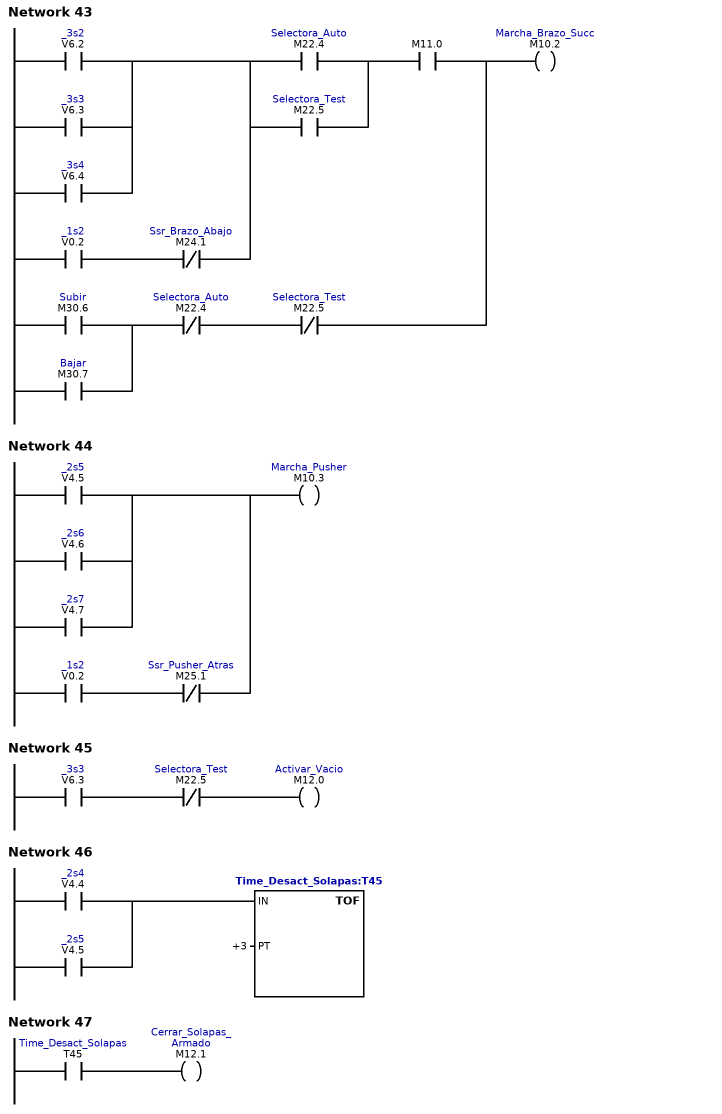
[picture p24: SBR6 networks 43-47]
Network 43
LD     _3s2:V6.2
O      _3s3:V6.3
O      _3s4:V6.4
LD     _1s2:V0.2
AN     Ssr_Brazo_Abajo:M24.1
OLD
LD     Selectora_Auto:M22.4
O      Selectora_Test:M22.5
ALD
A      M11.0
LD     Subir:M30.6
O      Bajar:M30.7
AN     Selectora_Auto:M22.4
AN     Selectora_Test:M22.5
OLD
=      Marcha_Brazo_Succ:M10.2
Network 44
LD     _2s5:V4.5
O      _2s6:V4.6
O      _2s7:V4.7
LD     _1s2:V0.2
AN     Ssr_Pusher_Atras:M25.1
OLD
=      Marcha_Pusher:M10.3
Network 45
LD     _3s3:V6.3
AN     Selectora_Test:M22.5
=      Activar_Vacio:M12.0
Network 46
LD     _2s4:V4.4
O      _2s5:V4.5
TOF    Time_Desact_Solapas:T45, +3
Network 47
LD     Time_Desact_Solapas:T45
=      Cerrar_Solapas_Armado:M12.1
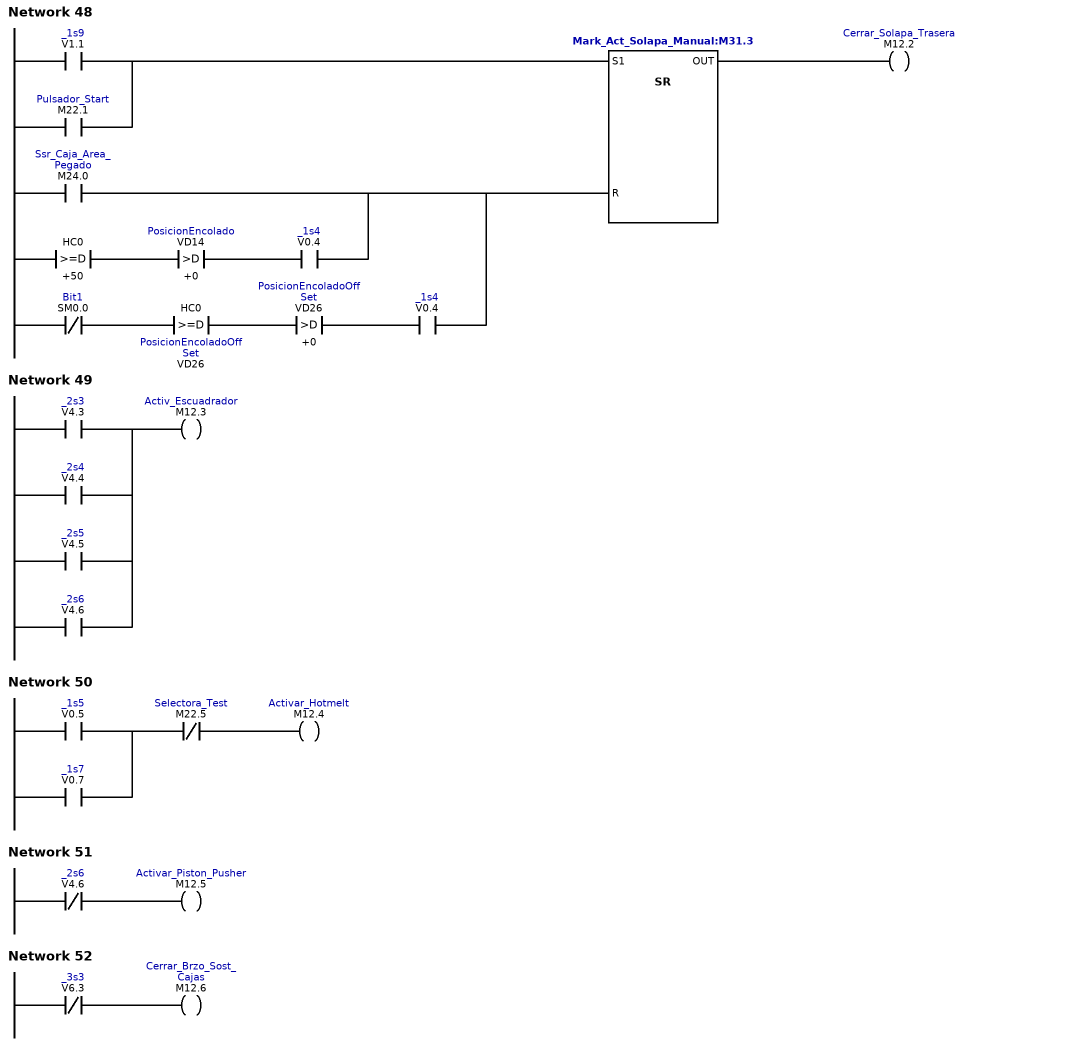
Network 48
LD     _1s9:V1.1
O      Pulsador_Start:M22.1
LD     Ssr_Caja_Area_Pegado:M24.0
LDD>=  HC0, +50
AD>    PosicionEncolado:VD14, +0
A      _1s4:V0.4
OLD
LDN    Bit1:SM0.0
AD>=   HC0, PosicionEncoladoOffSet:VD26
AD>    PosicionEncoladoOffSet:VD26, +0
A      _1s4:V0.4
OLD
NOT
A      Mark_Act_Solapa_Manual:M31.3
OLD
=      Mark_Act_Solapa_Manual:M31.3
=      Cerrar_Solapa_Trasera:M12.2
Network 49
LD     _2s3:V4.3
O      _2s4:V4.4
O      _2s5:V4.5
O      _2s6:V4.6
=      Activ_Escuadrador:M12.3
Network 50
LD     _1s5:V0.5
O      _1s7:V0.7
AN     Selectora_Test:M22.5
=      Activar_Hotmelt:M12.4
Network 51
LDN    _2s6:V4.6
=      Activar_Piston_Pusher:M12.5
Network 52
LDN    _3s3:V6.3
=      Cerrar_Brzo_Sost_Cajas:M12.6
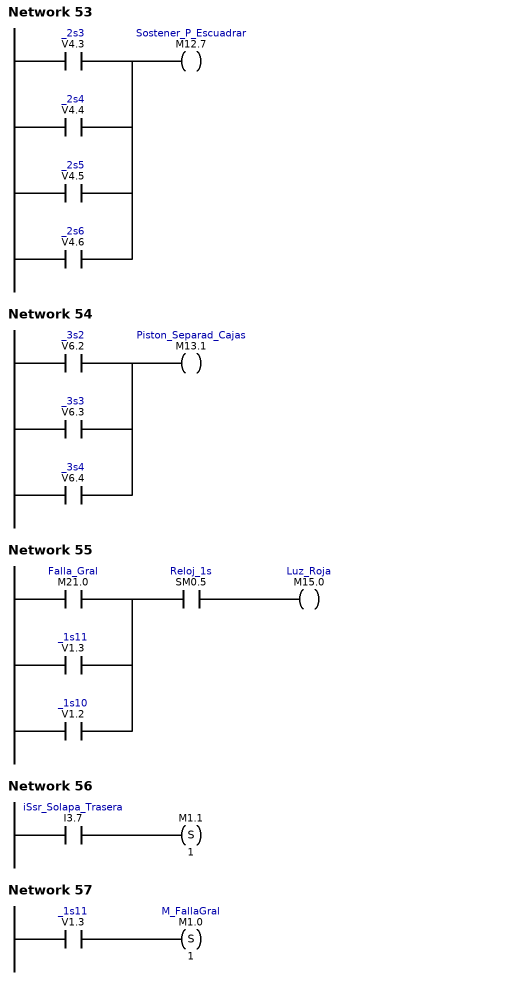
Network 53
LD     _2s3:V4.3
O      _2s4:V4.4
O      _2s5:V4.5
O      _2s6:V4.6
=      Sostener_P_Escuadrar:M12.7
Network 54
LD     _3s2:V6.2
O      _3s3:V6.3
O      _3s4:V6.4
=      Piston_Separad_Cajas:M13.1
Network 55
LD     Falla_Gral:M21.0
O      _1s11:V1.3
O      _1s10:V1.2
A      Reloj_1s:SM0.5
=      Luz_Roja:M15.0
Network 56
LD     iSsr_Solapa_Trasera:I3.7
S      M1.1, 1
Network 57
LD     _1s11:V1.3
S      M_FallaGral:M1.0, 1
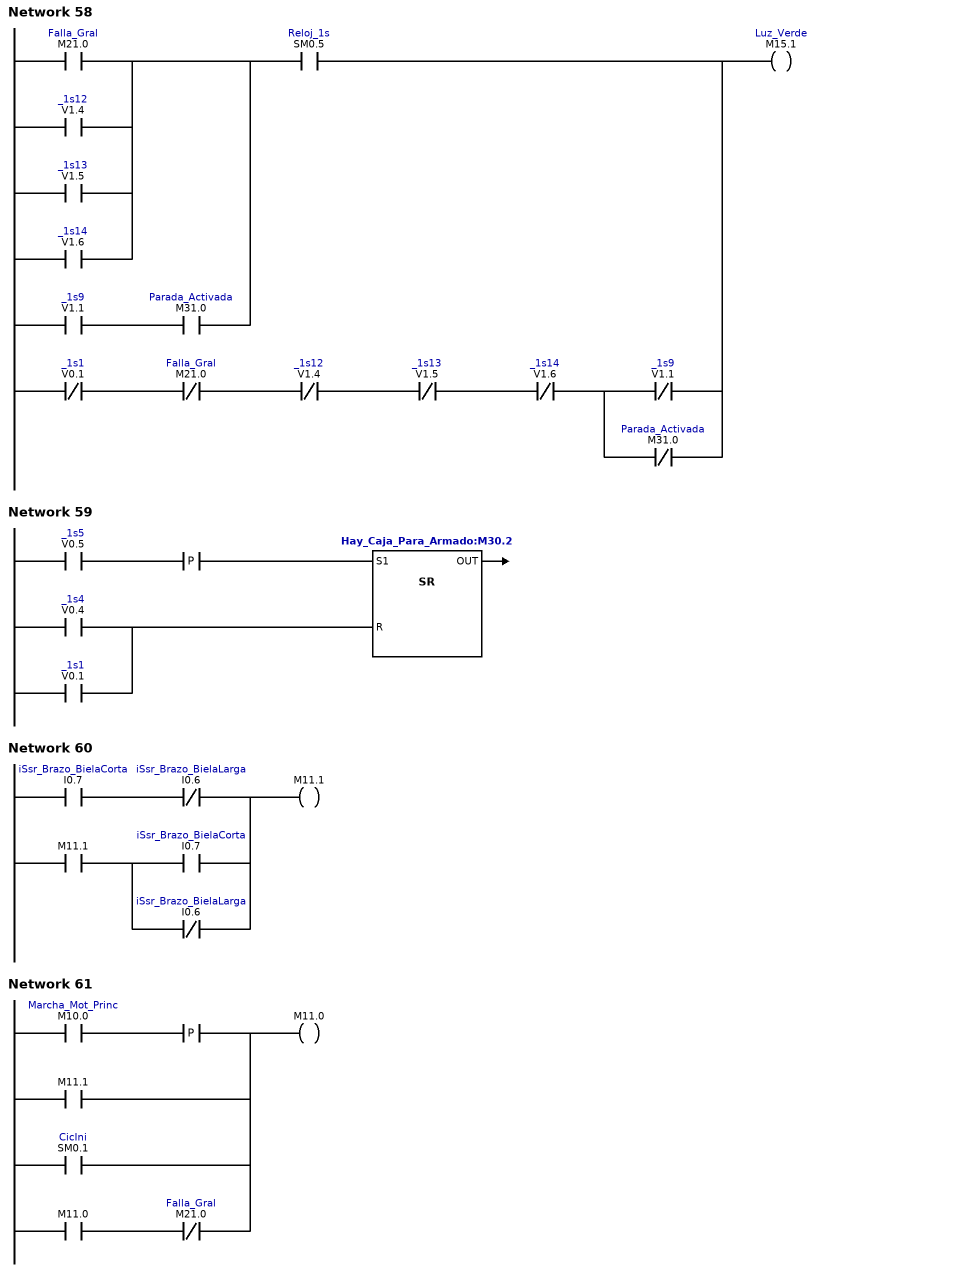
Network 58
LD     Falla_Gral:M21.0
O      _1s12:V1.4
O      _1s13:V1.5
O      _1s14:V1.6
LD     _1s9:V1.1
A      Parada_Activada:M31.0
OLD
A      Reloj_1s:SM0.5
LDN    _1s1:V0.1
AN     Falla_Gral:M21.0
AN     _1s12:V1.4
AN     _1s13:V1.5
AN     _1s14:V1.6
LDN    _1s9:V1.1
ON     Parada_Activada:M31.0
ALD
OLD
=      Luz_Verde:M15.1
Network 59
LD     _1s5:V0.5
EU
LD     _1s4:V0.4
O      _1s1:V0.1
NOT
A      Hay_Caja_Para_Armado:M30.2
OLD
=      Hay_Caja_Para_Armado:M30.2
Network 60
LD     iSsr_Brazo_BielaCorta:I0.7
AN     iSsr_Brazo_BielaLarga:I0.6
LD     M11.1
LD     iSsr_Brazo_BielaCorta:I0.7
ON     iSsr_Brazo_BielaLarga:I0.6
ALD
OLD
=      M11.1
Network 61
LD     Marcha_Mot_Princ:M10.0
EU
O      M11.1
O      CicIni:SM0.1
LD     M11.0
AN     Falla_Gral:M21.0
OLD
=      M11.0
END_SUBROUTINE_BLOCK

SUBROUTINE_BLOCK Secuencial_2:SBR7
TITLE=
BEGIN
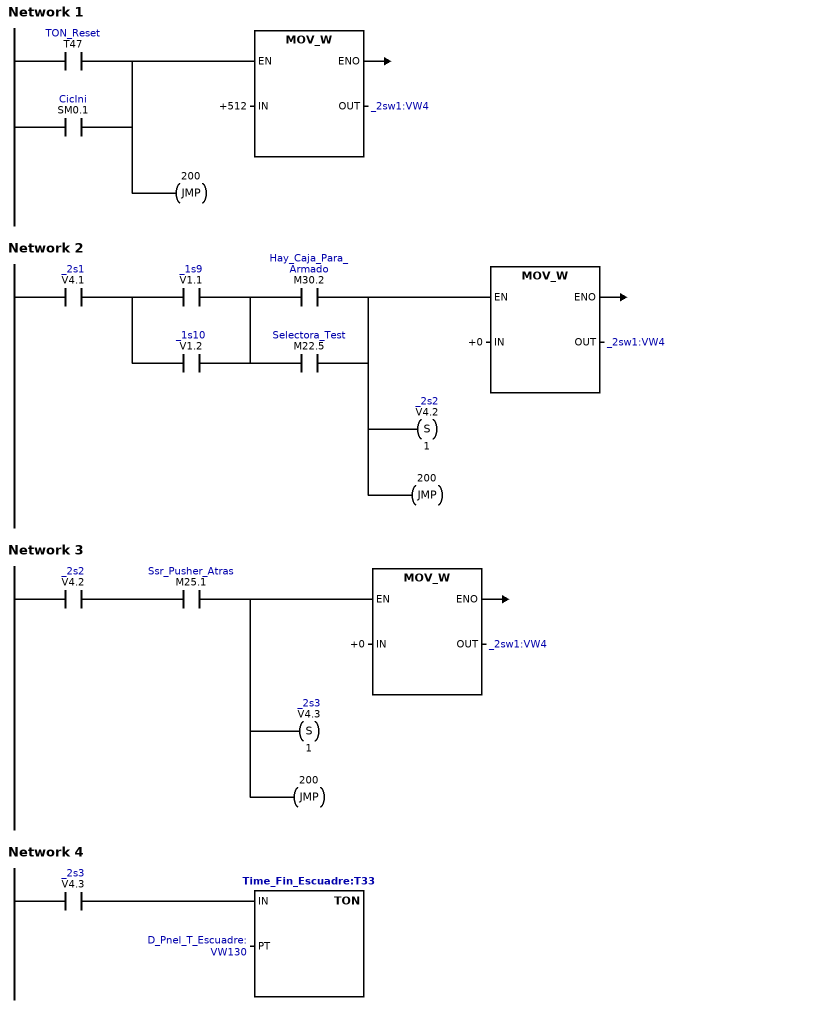
Network 1
LD     TON_Reset:T47
O      CicIni:SM0.1
MOVW   +512, _2sw1:VW4
JMP    200
Network 2
LD     _2s1:V4.1
LD     _1s9:V1.1
O      _1s10:V1.2
ALD
LD     Hay_Caja_Para_Armado:M30.2
O      Selectora_Test:M22.5
ALD
MOVW   +0, _2sw1:VW4
S      _2s2:V4.2, 1
JMP    200
Network 3
LD     _2s2:V4.2
A      Ssr_Pusher_Atras:M25.1
MOVW   +0, _2sw1:VW4
S      _2s3:V4.3, 1
JMP    200
Network 4
LD     _2s3:V4.3
TON    Time_Fin_Escuadre:T33, D_Pnel_T_Escuadre:VW130
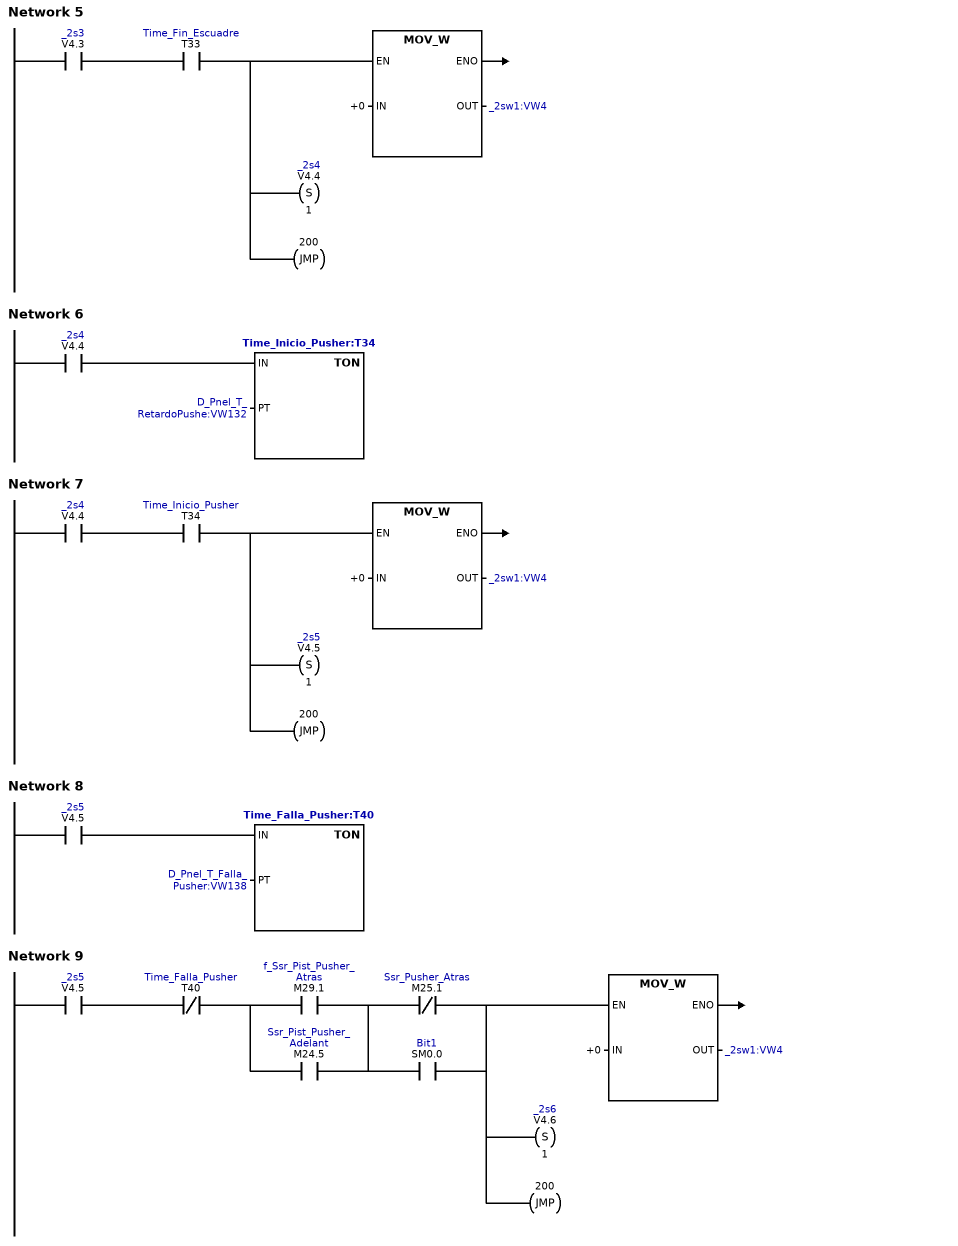
Network 5
LD     _2s3:V4.3
A      Time_Fin_Escuadre:T33
MOVW   +0, _2sw1:VW4
S      _2s4:V4.4, 1
JMP    200
Network 6
LD     _2s4:V4.4
TON    Time_Inicio_Pusher:T34, D_Pnel_T_RetardoPushe:VW132
Network 7
LD     _2s4:V4.4
A      Time_Inicio_Pusher:T34
MOVW   +0, _2sw1:VW4
S      _2s5:V4.5, 1
JMP    200
Network 8
LD     _2s5:V4.5
TON    Time_Falla_Pusher:T40, D_Pnel_T_Falla_Pusher:VW138
Network 9
LD     _2s5:V4.5
AN     Time_Falla_Pusher:T40
LD     f_Ssr_Pist_Pusher_Atras:M29.1
O      Ssr_Pist_Pusher_Adelant:M24.5
ALD
LDN    Ssr_Pusher_Atras:M25.1
O      Bit1:SM0.0
ALD
MOVW   +0, _2sw1:VW4
S      _2s6:V4.6, 1
JMP    200
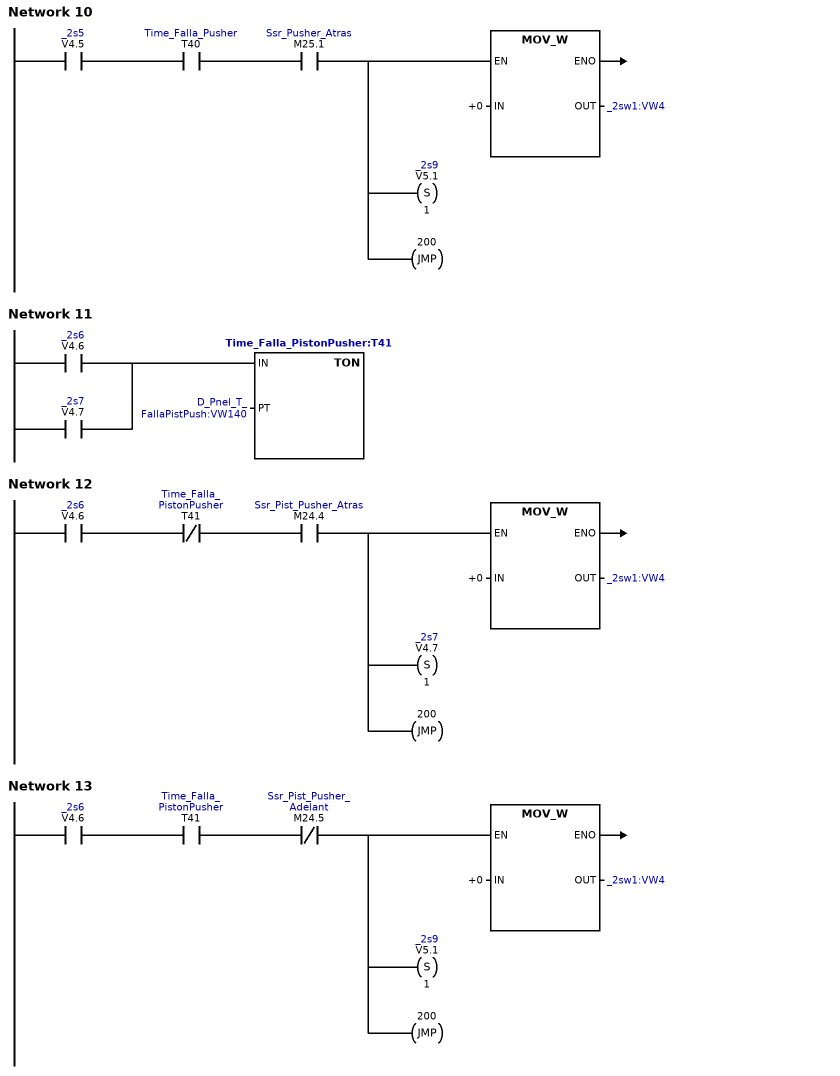
Network 10
LD     _2s5:V4.5
A      Time_Falla_Pusher:T40
A      Ssr_Pusher_Atras:M25.1
MOVW   +0, _2sw1:VW4
S      _2s9:V5.1, 1
JMP    200
Network 11
LD     _2s6:V4.6
O      _2s7:V4.7
TON    Time_Falla_PistonPusher:T41, D_Pnel_T_FallaPistPush:VW140
Network 12
LD     _2s6:V4.6
AN     Time_Falla_PistonPusher:T41
A      Ssr_Pist_Pusher_Atras:M24.4
MOVW   +0, _2sw1:VW4
S      _2s7:V4.7, 1
JMP    200
Network 13
LD     _2s6:V4.6
A      Time_Falla_PistonPusher:T41
AN     Ssr_Pist_Pusher_Adelant:M24.5
MOVW   +0, _2sw1:VW4
S      _2s9:V5.1, 1
JMP    200
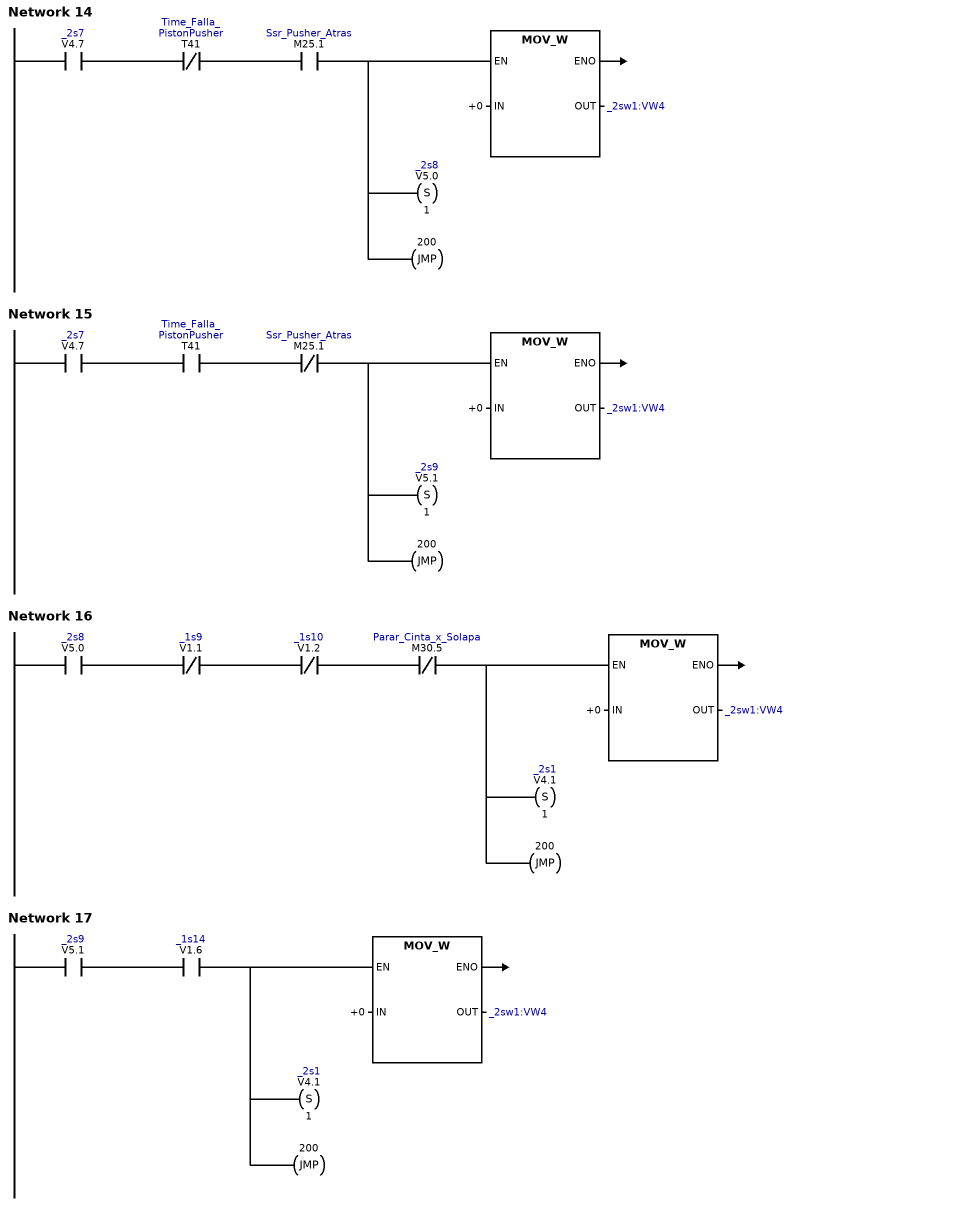
Network 14
LD     _2s7:V4.7
AN     Time_Falla_PistonPusher:T41
A      Ssr_Pusher_Atras:M25.1
MOVW   +0, _2sw1:VW4
S      _2s8:V5.0, 1
JMP    200
Network 15
LD     _2s7:V4.7
A      Time_Falla_PistonPusher:T41
AN     Ssr_Pusher_Atras:M25.1
MOVW   +0, _2sw1:VW4
S      _2s9:V5.1, 1
JMP    200
Network 16
LD     _2s8:V5.0
AN     _1s9:V1.1
AN     _1s10:V1.2
AN     Parar_Cinta_x_Solapa:M30.5
MOVW   +0, _2sw1:VW4
S      _2s1:V4.1, 1
JMP    200
Network 17
LD     _2s9:V5.1
A      _1s14:V1.6
MOVW   +0, _2sw1:VW4
S      _2s1:V4.1, 1
JMP    200
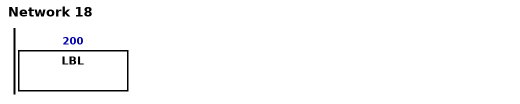
Network 18
LBL    200
END_SUBROUTINE_BLOCK

SUBROUTINE_BLOCK Secuencial_3:SBR8
TITLE=
BEGIN
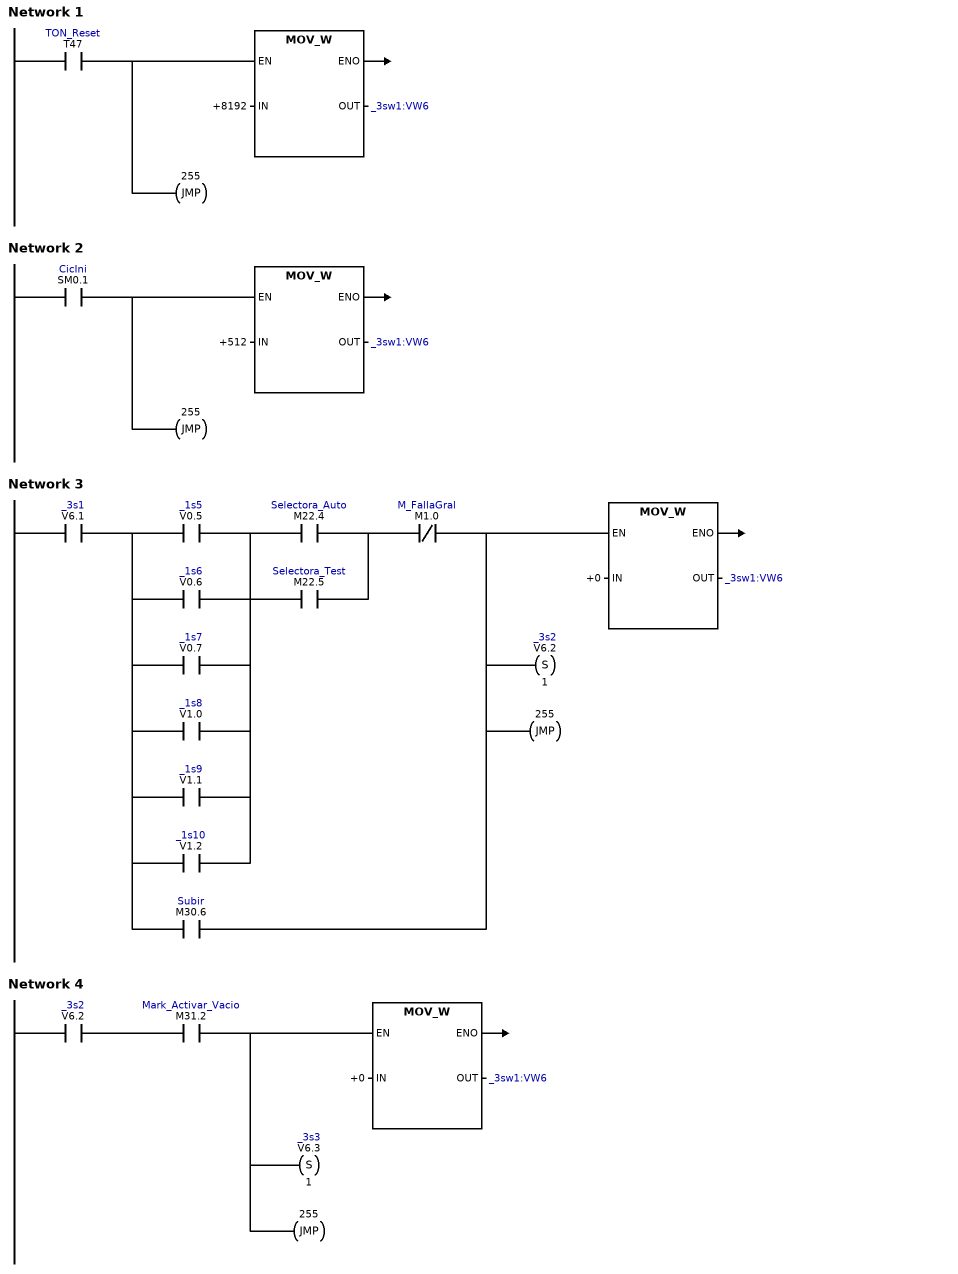
Network 1
LD     TON_Reset:T47
MOVW   +8192, _3sw1:VW6
JMP    255
Network 2
LD     CicIni:SM0.1
MOVW   +512, _3sw1:VW6
JMP    255
Network 3
LD     _3s1:V6.1
LD     _1s5:V0.5
O      _1s6:V0.6
O      _1s7:V0.7
O      _1s8:V1.0
O      _1s9:V1.1
O      _1s10:V1.2
LD     Selectora_Auto:M22.4
O      Selectora_Test:M22.5
ALD
AN     M_FallaGral:M1.0
O      Subir:M30.6
ALD
MOVW   +0, _3sw1:VW6
S      _3s2:V6.2, 1
JMP    255
Network 4
LD     _3s2:V6.2
A      Mark_Activar_Vacio:M31.2
MOVW   +0, _3sw1:VW6
S      _3s3:V6.3, 1
JMP    255
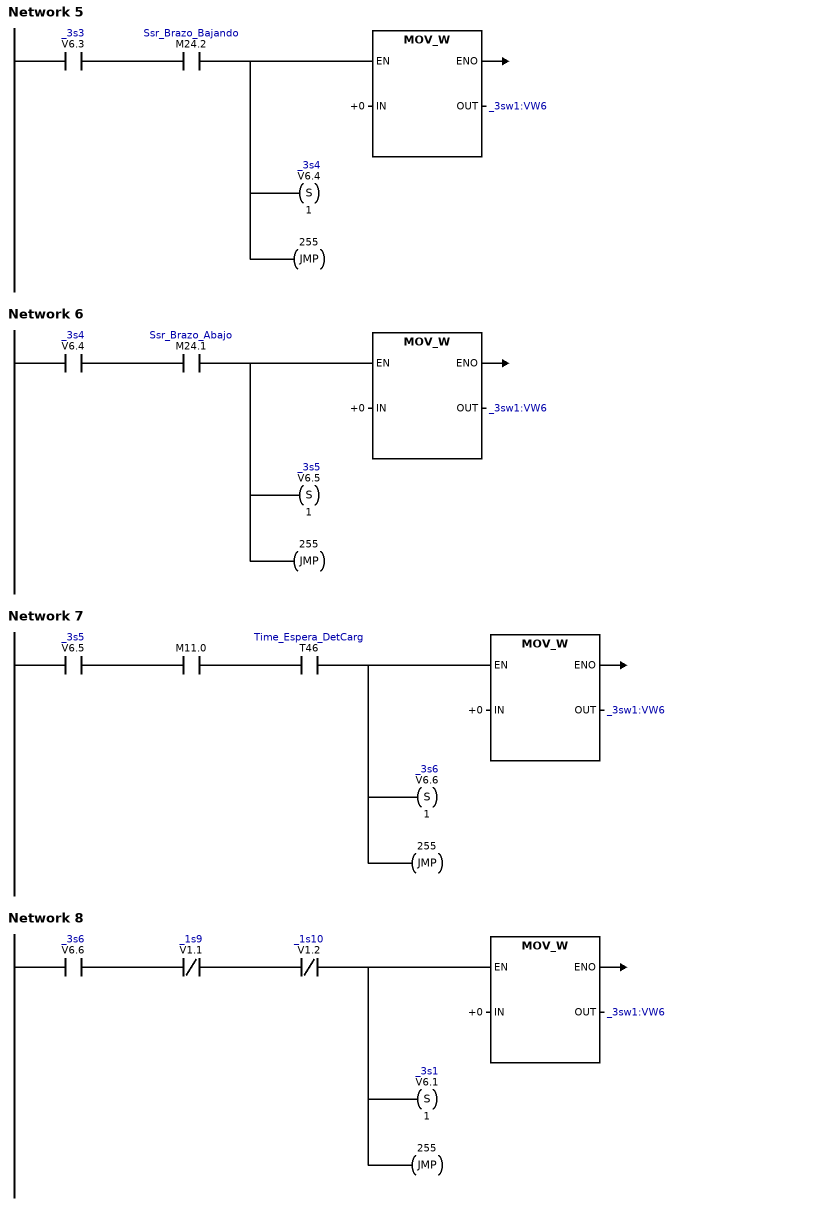
Network 5
LD     _3s3:V6.3
A      Ssr_Brazo_Bajando:M24.2
MOVW   +0, _3sw1:VW6
S      _3s4:V6.4, 1
JMP    255
Network 6
LD     _3s4:V6.4
A      Ssr_Brazo_Abajo:M24.1
MOVW   +0, _3sw1:VW6
S      _3s5:V6.5, 1
JMP    255
Network 7
LD     _3s5:V6.5
A      M11.0
A      Time_Espera_DetCarg:T46
MOVW   +0, _3sw1:VW6
S      _3s6:V6.6, 1
JMP    255
Network 8
LD     _3s6:V6.6
AN     _1s9:V1.1
AN     _1s10:V1.2
MOVW   +0, _3sw1:VW6
S      _3s1:V6.1, 1
JMP    255
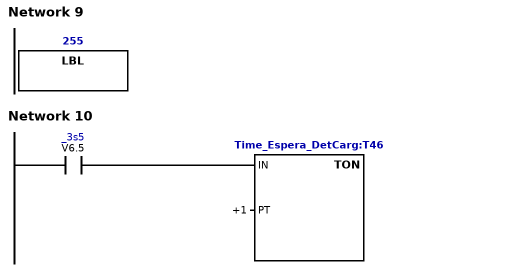
Network 9
LBL    255
Network 10
LD     _3s5:V6.5
TON    Time_Espera_DetCarg:T46, +1
END_SUBROUTINE_BLOCK

SUBROUTINE_BLOCK Subir_Bajar_Brazo:SBR13
TITLE=
BEGIN
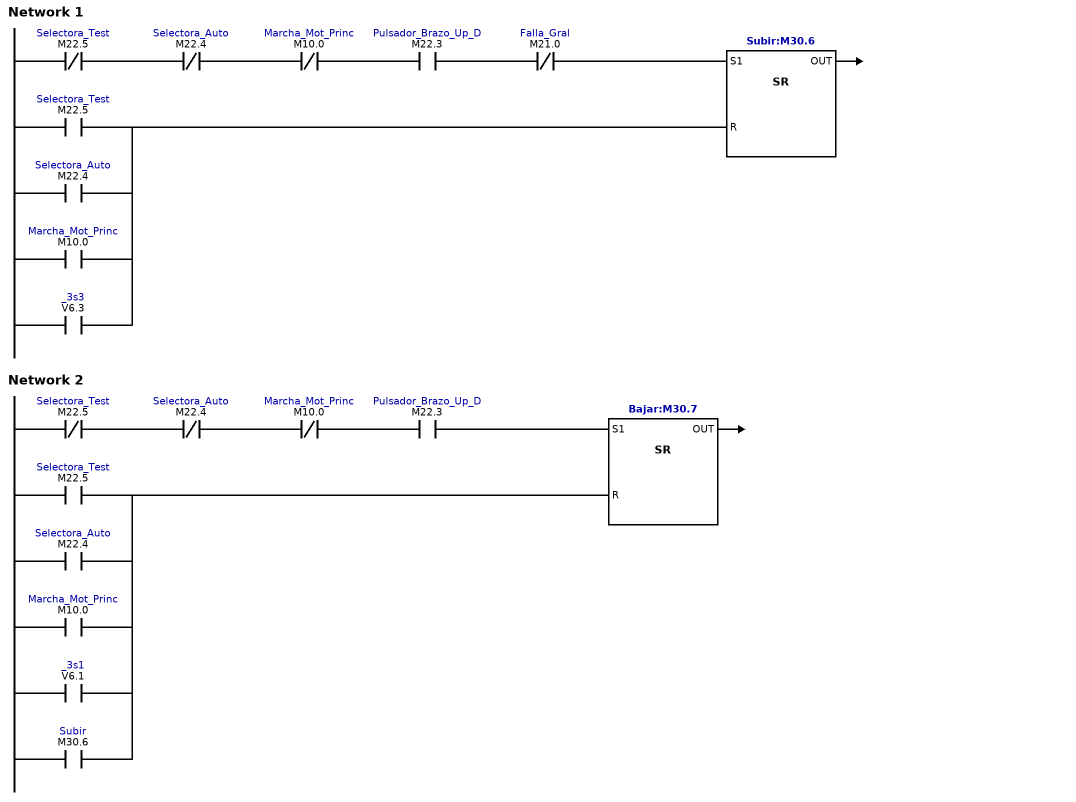
Network 1
LDN    Selectora_Test:M22.5
AN     Selectora_Auto:M22.4
AN     Marcha_Mot_Princ:M10.0
A      Pulsador_Brazo_Up_D:M22.3
AN     Falla_Gral:M21.0
LD     Selectora_Test:M22.5
O      Selectora_Auto:M22.4
O      Marcha_Mot_Princ:M10.0
O      _3s3:V6.3
NOT
A      Subir:M30.6
OLD
=      Subir:M30.6
Network 2
LDN    Selectora_Test:M22.5
AN     Selectora_Auto:M22.4
AN     Marcha_Mot_Princ:M10.0
A      Pulsador_Brazo_Up_D:M22.3
LD     Selectora_Test:M22.5
O      Selectora_Auto:M22.4
O      Marcha_Mot_Princ:M10.0
O      _3s1:V6.1
O      Subir:M30.6
NOT
A      Bajar:M30.7
OLD
=      Bajar:M30.7
END_SUBROUTINE_BLOCK

SUBROUTINE_BLOCK Tratado_Alarmas:SBR14
TITLE=
BEGIN
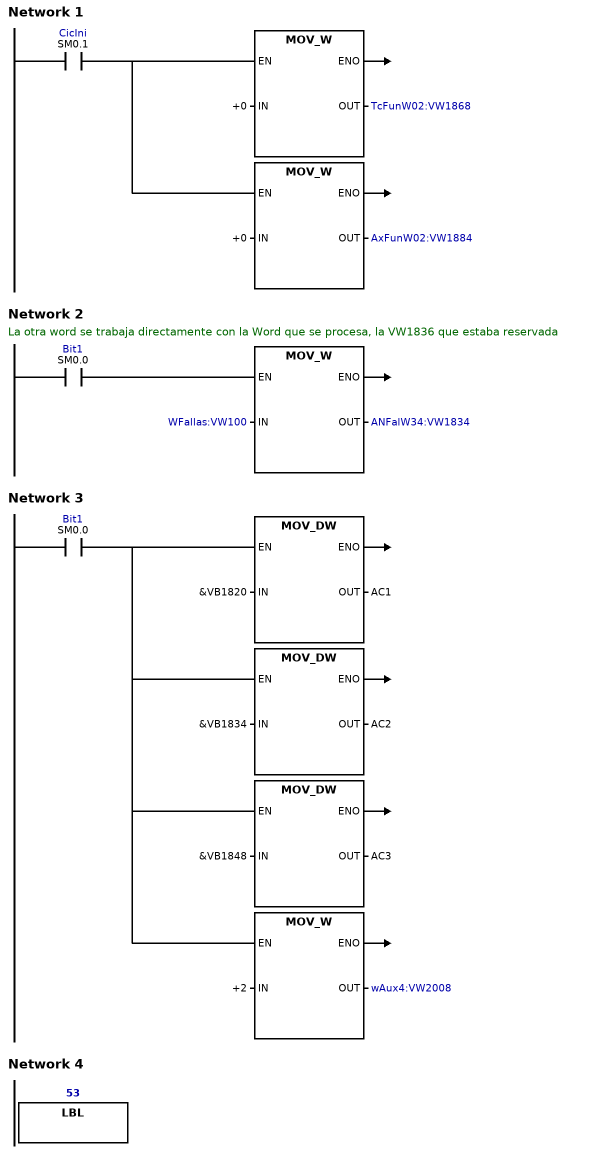
Network 1
LD     CicIni:SM0.1
MOVW   +0, TcFunW02:VW1868
MOVW   +0, AxFunW02:VW1884
Network 2
// La otra word se trabaja directamente con la Word que se procesa, la VW1836 que estaba reservada
LD     Bit1:SM0.0
MOVW   WFallas:VW100, ANFalW34:VW1834
Network 3
LD     Bit1:SM0.0
MOVD   &VB1820, AC1
MOVD   &VB1834, AC2
MOVD   &VB1848, AC3
MOVW   +2, wAux4:VW2008
Network 4
LBL    53
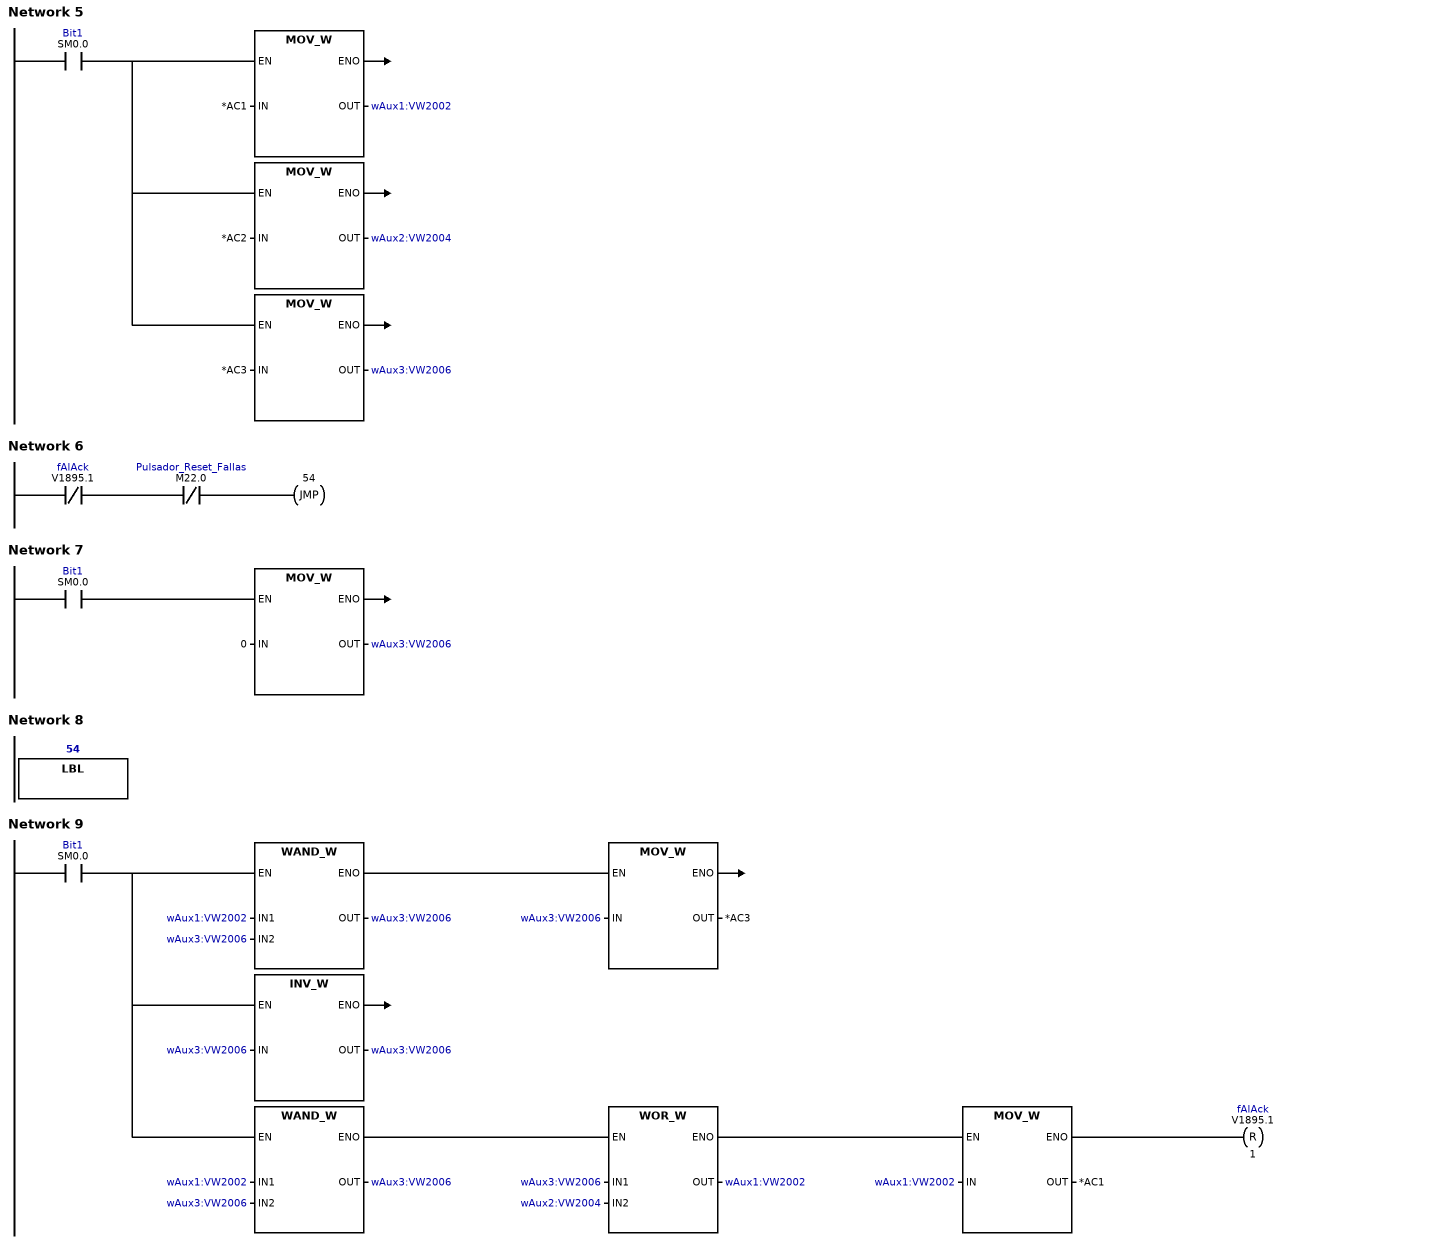
Network 5
LD     Bit1:SM0.0
MOVW   *AC1, wAux1:VW2002
MOVW   *AC2, wAux2:VW2004
MOVW   *AC3, wAux3:VW2006
Network 6
LDN    fAlAck:V1895.1
AN     Pulsador_Reset_Fallas:M22.0
JMP    54
Network 7
LD     Bit1:SM0.0
MOVW   0, wAux3:VW2006
Network 8
LBL    54
Network 9
LD     Bit1:SM0.0
LPS
ANDW   wAux1:VW2002, wAux3:VW2006
AENO
MOVW   wAux3:VW2006, *AC3
LRD
INVW   wAux3:VW2006
LPP
ANDW   wAux1:VW2002, wAux3:VW2006
AENO
MOVW   wAux3:VW2006, wAux1:VW2002
AENO
ORW    wAux2:VW2004, wAux1:VW2002
AENO
MOVW   wAux1:VW2002, *AC1
AENO
R      fAlAck:V1895.1, 1
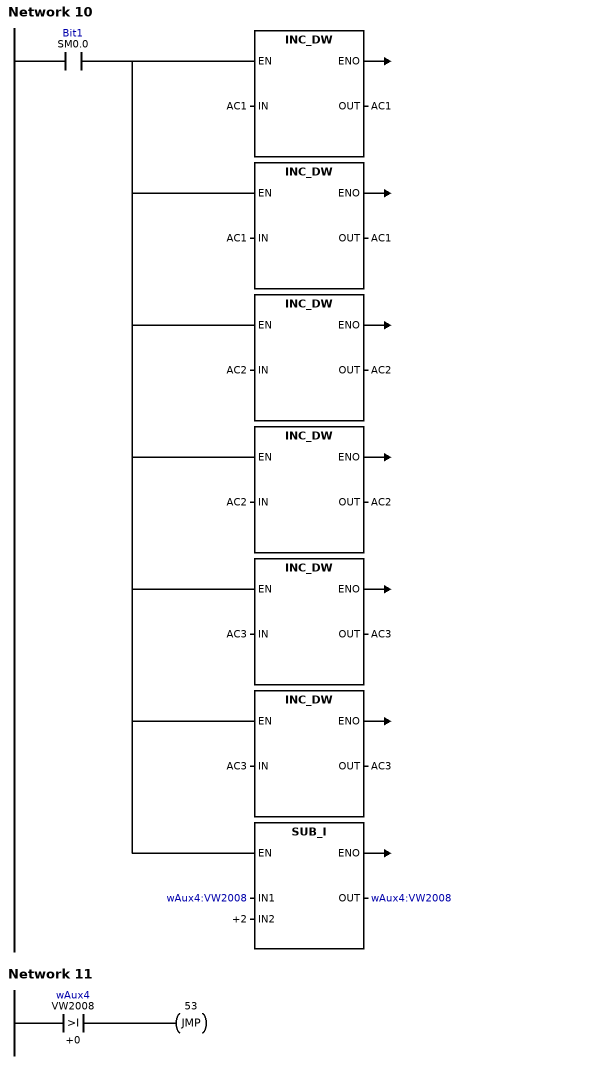
Network 10
LD     Bit1:SM0.0
INCD   AC1
INCD   AC1
INCD   AC2
INCD   AC2
INCD   AC3
INCD   AC3
-I     +2, wAux4:VW2008
Network 11
LDW>   wAux4:VW2008, +0
JMP    53
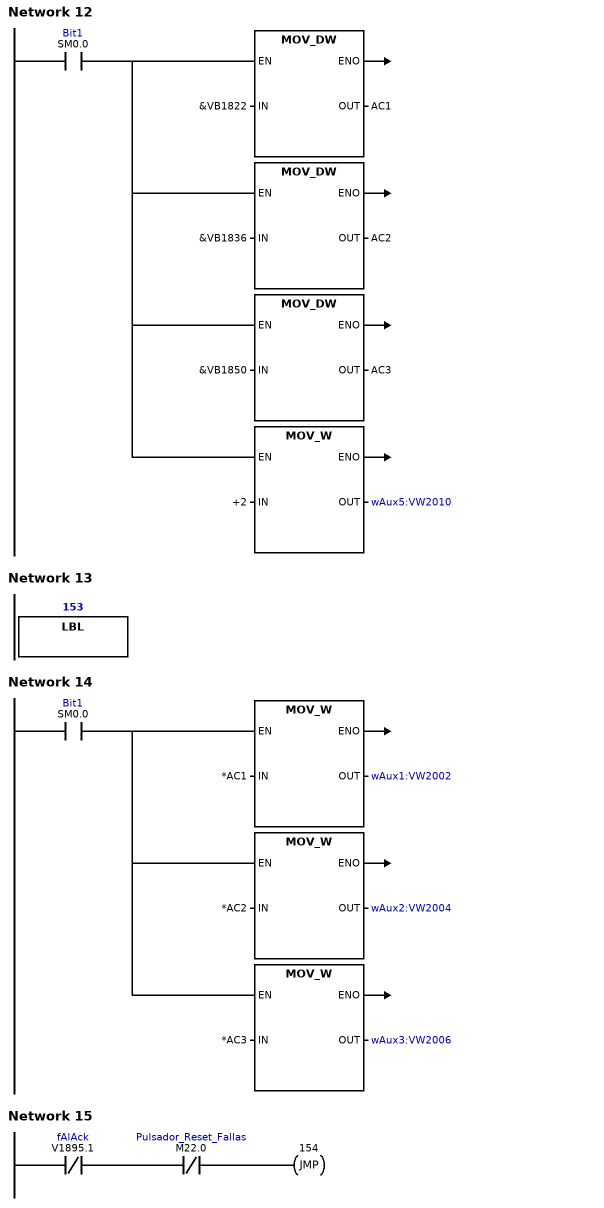
Network 12
LD     Bit1:SM0.0
MOVD   &VB1822, AC1
MOVD   &VB1836, AC2
MOVD   &VB1850, AC3
MOVW   +2, wAux5:VW2010
Network 13
LBL    153
Network 14
LD     Bit1:SM0.0
MOVW   *AC1, wAux1:VW2002
MOVW   *AC2, wAux2:VW2004
MOVW   *AC3, wAux3:VW2006
Network 15
LDN    fAlAck:V1895.1
AN     Pulsador_Reset_Fallas:M22.0
JMP    154
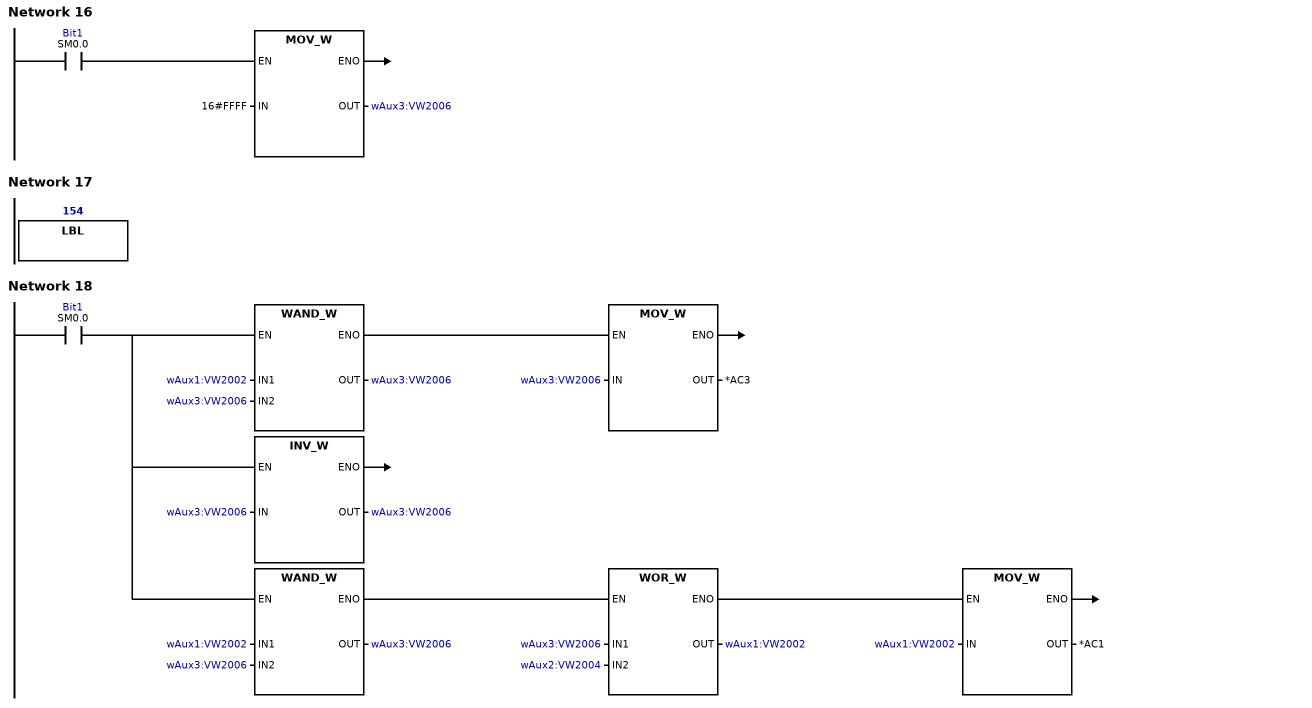
Network 16
LD     Bit1:SM0.0
MOVW   16#FFFF, wAux3:VW2006
Network 17
LBL    154
Network 18
LD     Bit1:SM0.0
LPS
ANDW   wAux1:VW2002, wAux3:VW2006
AENO
MOVW   wAux3:VW2006, *AC3
LRD
INVW   wAux3:VW2006
LPP
ANDW   wAux1:VW2002, wAux3:VW2006
AENO
MOVW   wAux3:VW2006, wAux1:VW2002
AENO
ORW    wAux2:VW2004, wAux1:VW2002
AENO
MOVW   wAux1:VW2002, *AC1
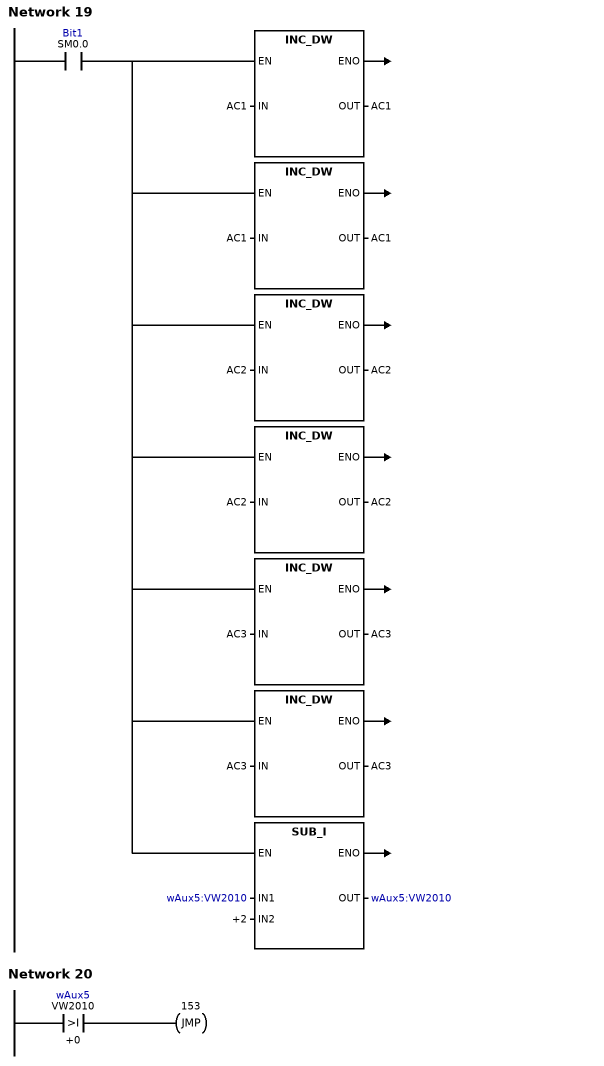
Network 19
LD     Bit1:SM0.0
INCD   AC1
INCD   AC1
INCD   AC2
INCD   AC2
INCD   AC3
INCD   AC3
-I     +2, wAux5:VW2010
Network 20
LDW>   wAux5:VW2010, +0
JMP    153
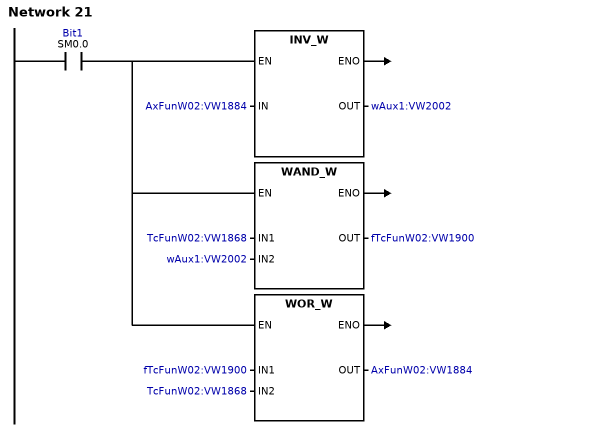
Network 21
LD     Bit1:SM0.0
MOVW   AxFunW02:VW1884, wAux1:VW2002
INVW   wAux1:VW2002
MOVW   TcFunW02:VW1868, fTcFunW02:VW1900
ANDW   wAux1:VW2002, fTcFunW02:VW1900
MOVW   fTcFunW02:VW1900, AxFunW02:VW1884
ORW    TcFunW02:VW1868, AxFunW02:VW1884
END_SUBROUTINE_BLOCK

SUBROUTINE_BLOCK Fallas:SBR20
TITLE=
BEGIN
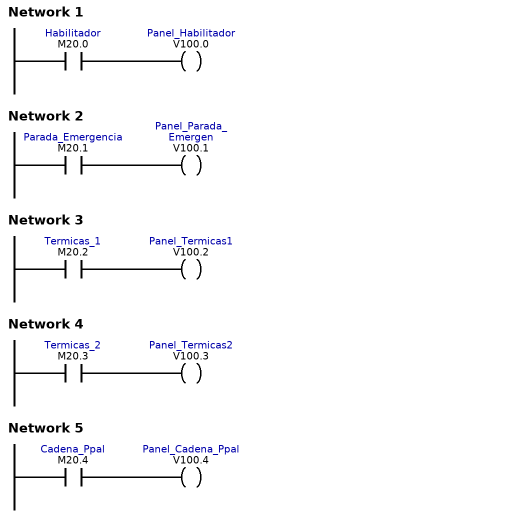
Network 1
LD     Habilitador:M20.0
=      Panel_Habilitador:V100.0
Network 2
LD     Parada_Emergencia:M20.1
=      Panel_Parada_Emergen:V100.1
Network 3
LD     Termicas_1:M20.2
=      Panel_Termicas1:V100.2
Network 4
LD     Termicas_2:M20.3
=      Panel_Termicas2:V100.3
Network 5
LD     Cadena_Ppal:M20.4
=      Panel_Cadena_Ppal:V100.4
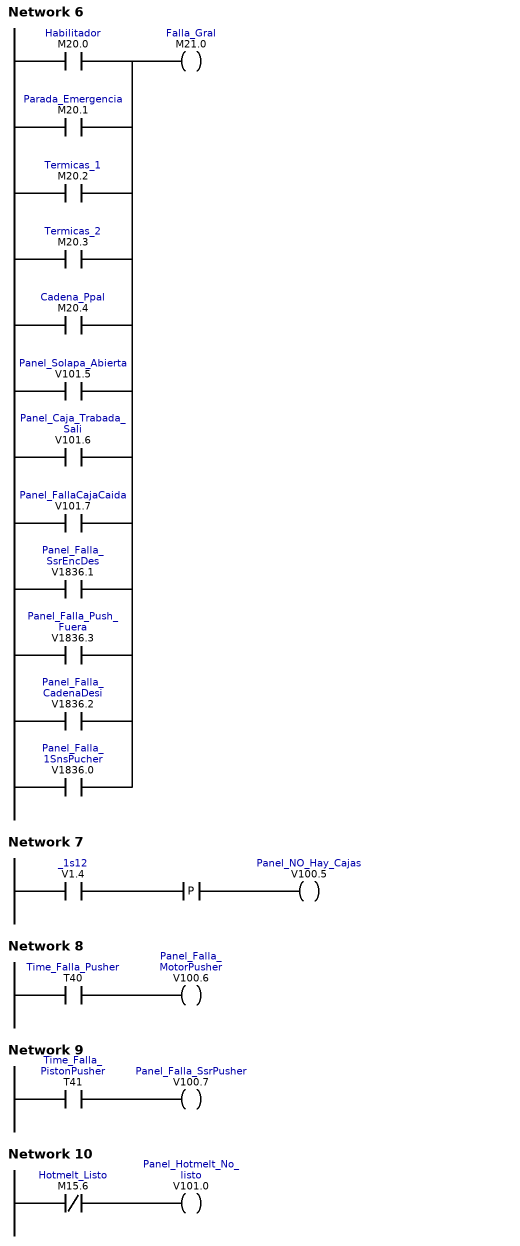
Network 6
LD     Habilitador:M20.0
O      Parada_Emergencia:M20.1
O      Termicas_1:M20.2
O      Termicas_2:M20.3
O      Cadena_Ppal:M20.4
O      Panel_Solapa_Abierta:V101.5
O      Panel_Caja_Trabada_Sali:V101.6
O      Panel_FallaCajaCaida:V101.7
O      Panel_Falla_SsrEncDes:V1836.1
O      Panel_Falla_Push_Fuera:V1836.3
O      Panel_Falla_CadenaDesi:V1836.2
O      Panel_Falla_1SnsPucher:V1836.0
=      Falla_Gral:M21.0
Network 7
LD     _1s12:V1.4
EU
=      Panel_NO_Hay_Cajas:V100.5
Network 8
LD     Time_Falla_Pusher:T40
=      Panel_Falla_MotorPusher:V100.6
Network 9
LD     Time_Falla_PistonPusher:T41
=      Panel_Falla_SsrPusher:V100.7
Network 10
LDN    Hotmelt_Listo:M15.6
=      Panel_Hotmelt_No_listo:V101.0
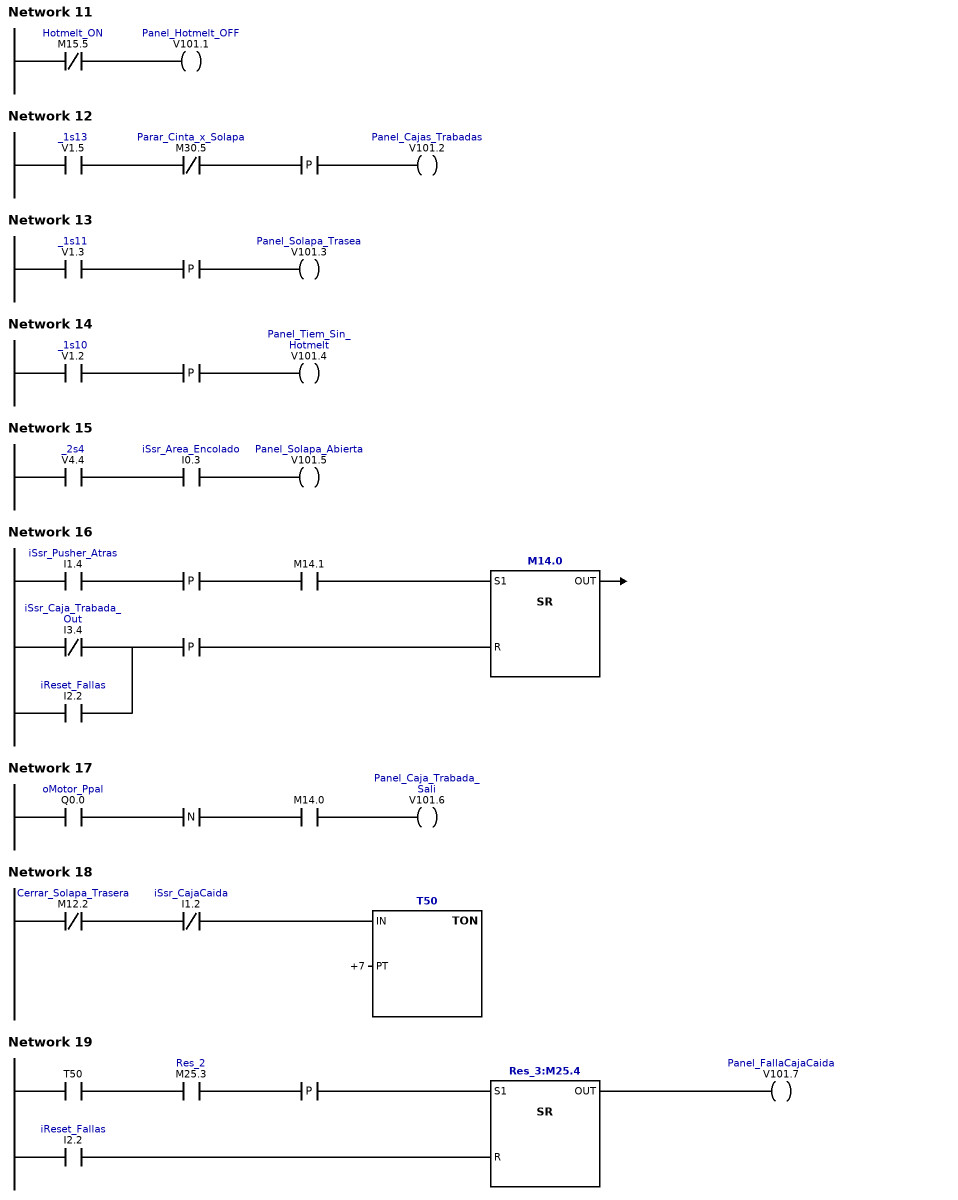
Network 11
LDN    Hotmelt_ON:M15.5
=      Panel_Hotmelt_OFF:V101.1
Network 12
LD     _1s13:V1.5
AN     Parar_Cinta_x_Solapa:M30.5
EU
=      Panel_Cajas_Trabadas:V101.2
Network 13
LD     _1s11:V1.3
EU
=      Panel_Solapa_Trasea:V101.3
Network 14
LD     _1s10:V1.2
EU
=      Panel_Tiem_Sin_Hotmelt:V101.4
Network 15
LD     _2s4:V4.4
A      iSsr_Area_Encolado:I0.3
=      Panel_Solapa_Abierta:V101.5
Network 16
LD     iSsr_Pusher_Atras:I1.4
EU
A      M14.1
LDN    iSsr_Caja_Trabada_Out:I3.4
O      iReset_Fallas:I2.2
EU
NOT
A      M14.0
OLD
=      M14.0
Network 17
LD     oMotor_Ppal:Q0.0
ED
A      M14.0
=      Panel_Caja_Trabada_Sali:V101.6
Network 18
LDN    Cerrar_Solapa_Trasera:M12.2
AN     iSsr_CajaCaida:I1.2
TON    T50, +7
Network 19
LD     T50
A      Res_2:M25.3
EU
LD     iReset_Fallas:I2.2
NOT
A      Res_3:M25.4
OLD
=      Res_3:M25.4
=      Panel_FallaCajaCaida:V101.7
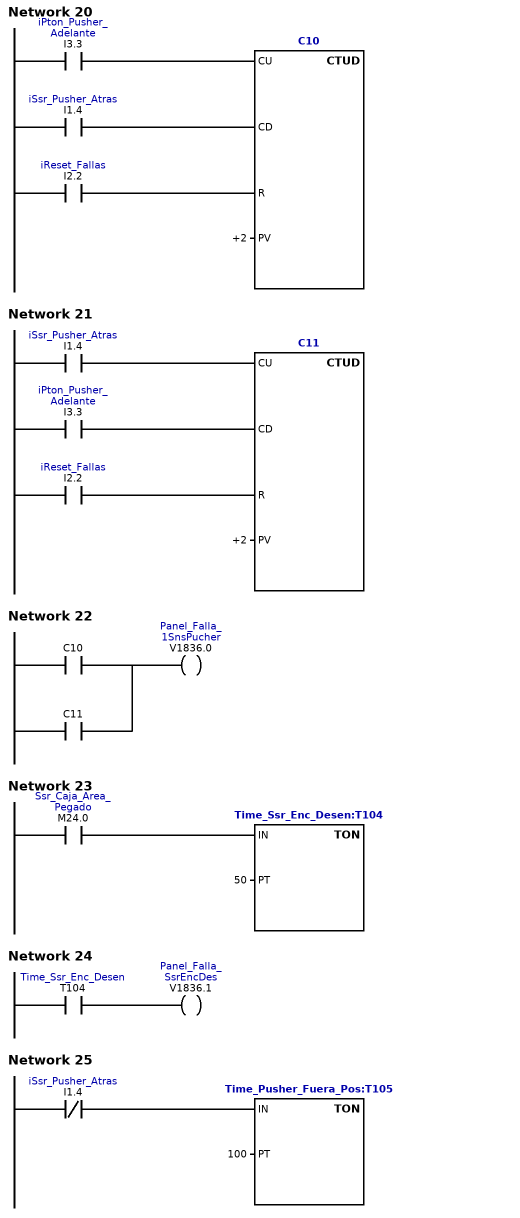
Network 20
LD     iPton_Pusher_Adelante:I3.3
LD     iSsr_Pusher_Atras:I1.4
LD     iReset_Fallas:I2.2
CTUD   C10, +2
Network 21
LD     iSsr_Pusher_Atras:I1.4
LD     iPton_Pusher_Adelante:I3.3
LD     iReset_Fallas:I2.2
CTUD   C11, +2
Network 22
LD     C10
O      C11
=      Panel_Falla_1SnsPucher:V1836.0
Network 23
LD     Ssr_Caja_Area_Pegado:M24.0
TON    Time_Ssr_Enc_Desen:T104, 50
Network 24
LD     Time_Ssr_Enc_Desen:T104
=      Panel_Falla_SsrEncDes:V1836.1
Network 25
LDN    iSsr_Pusher_Atras:I1.4
TON    Time_Pusher_Fuera_Pos:T105, 100
